// TIA Portal V20 export
FUNCTION_BLOCK "LConSMC_LevelControl"   // FB32023, SCL
// Dieser Funktionsbaustein überwacht einen Eingabewert (x), um zu erkennen ob er einen parametrierten Wert verletzt (überschreitet, unterschreitet). Der Funktionsbaustein kann in jedem zyklischen Interrupt aufgerufen werden.  Funktionsbaustein-ID: 0104 / Limit value monitor. The function block can be called in any cyclic task.  Function block ID: 0104
// stored: Access Published, IsIECCheckEnabled true, MemoryReserve 100, SetENOAutomatically true
   VAR_INPUT
      run { ExternalAccessible := 'False'; ExternalVisible := 'False'; ExternalWritable := 'False'} : Bool := FALSE;   // TRUE: Funktionsbaustein aktivieren / TRUE: Enable function block
      x { ExternalAccessible := 'False'; ExternalVisible := 'False'; ExternalWritable := 'False'} : LReal := 0.0;   // Eingangswert / Input value
      alarmHigh { ExternalAccessible := 'False'; ExternalVisible := 'False'; ExternalWritable := 'False'} : LReal := 100.0;   // Alarm, oberer Grenzwert / Alarm, upper limit value
      warningHigh { ExternalAccessible := 'False'; ExternalVisible := 'False'; ExternalWritable := 'False'} : LReal := 80.0;   // Warnung, oberer Grenzwert / Warning, upper limit value
      warningLow { ExternalAccessible := 'False'; ExternalVisible := 'False'; ExternalWritable := 'False'} : LReal := -80.0;   // Warnung, unterer Grenzwert / Warning, lower limit value
      alarmLow { ExternalAccessible := 'False'; ExternalVisible := 'False'; ExternalWritable := 'False'} : LReal := -100.0;   // Alarm, unterer Grenzwert / Alarm, lower limit value
      hyst { ExternalAccessible := 'False'; ExternalVisible := 'False'; ExternalWritable := 'False'} : LReal := 0.0;   // Hysterese (Betrag wird verwendet) / Hysteresis (Absolute value is used)
      delayTime { ExternalAccessible := 'False'; ExternalVisible := 'False'; ExternalWritable := 'False'} : Time := T#3S;   // [s] Ausgangsverzögerungszeit Für einen Wert von 0 ist die Verzögerung deaktiviert / [ s ] Output delay time delayTime = 0, signal delay is disabled
   END_VAR
   VAR_OUTPUT
      busy { ExternalAccessible := 'False'; ExternalVisible := 'False'; ExternalWritable := 'False'} : Bool := FALSE;   // TRUE: Der Funktionsbaustein ist aktiv / TRUE: Function block is activated
      alarmUpperLimit { ExternalAccessible := 'False'; ExternalVisible := 'False'; ExternalWritable := 'False'} : Bool;   // TRUE: oberer Alarmwert überschritten / TRUE: Upper alarm limit value exceeded
      alarmLowerLimit { ExternalAccessible := 'False'; ExternalVisible := 'False'; ExternalWritable := 'False'} : Bool;   // TRUE: unterer Alarmwert überschritten / TRUE: Lower alarm limit value exceeded
      warningUpperLimit { ExternalAccessible := 'False'; ExternalVisible := 'False'; ExternalWritable := 'False'} : Bool := FALSE;   // TRUE: oberer Warnwert überschritten / TRUE: Upper warning limit value exceeded
      warningLowerLimit { ExternalAccessible := 'False'; ExternalVisible := 'False'; ExternalWritable := 'False'} : Bool := FALSE;   // TRUE: unterer Warnwert überschritten / TRUE: Lower warning limit value exceeded
   END_VAR
   VAR
      statAlarmUpperLimitSafe { ExternalAccessible := 'False'; ExternalVisible := 'False'; ExternalWritable := 'False'} : Bool := FALSE;
      statWarningUpperLimitSafe { ExternalAccessible := 'False'; ExternalVisible := 'False'; ExternalWritable := 'False'} : Bool := FALSE;
      statWarningLowerLimitSafe { ExternalAccessible := 'False'; ExternalVisible := 'False'; ExternalWritable := 'False'} : Bool := FALSE;
      statAlarmLowerLimitSafe { ExternalAccessible := 'False'; ExternalVisible := 'False'; ExternalWritable := 'False'} : Bool := FALSE;
      instTONalUp { ExternalAccessible := 'False'; ExternalVisible := 'False'; ExternalWritable := 'False'} : TON_TIME;
      instTONwaUp { ExternalAccessible := 'False'; ExternalVisible := 'False'; ExternalWritable := 'False'} : TON_TIME;
      instTONwaLo { ExternalAccessible := 'False'; ExternalVisible := 'False'; ExternalWritable := 'False'} : TON_TIME;
      instTONalLo { ExternalAccessible := 'False'; ExternalVisible := 'False'; ExternalWritable := 'False'} : TON_TIME;
      statAlarmUpperLimit { ExternalAccessible := 'False'; ExternalVisible := 'False'; ExternalWritable := 'False'} : Bool := FALSE;
      statAlarmLowerLimit { ExternalAccessible := 'False'; ExternalVisible := 'False'; ExternalWritable := 'False'} : Bool := FALSE;
      statWarningUpperLimit { ExternalAccessible := 'False'; ExternalVisible := 'False'; ExternalWritable := 'False'} : Bool := FALSE;
      statWarningLowerLimit { ExternalAccessible := 'False'; ExternalVisible := 'False'; ExternalWritable := 'False'} : Bool := FALSE;
   END_VAR
BEGIN
   REGION BLOCK INFO HEADER
     //===============================================================================
     // SIEMENS AG / (c)Copyright 2023
     //-------------------------------------------------------------------------------
     // Title:            LConSMC_LevelControl
     // Comment/Function: Limit value evaluation with warning level and alarm level
     // Library/Family:   LConSMC
     // Author:           APC Erlangen
     // Tested with:      FW 2.8
     // Engineering:      TIA Portal V16
     // Restrictions:     Needs to be called in a cyclic task
     // Requirements:     -
     //-------------------------------------------------------------------------------
     // Change log table:
     // Version  | Date       | Expert in charge       | Changes applied
     //----------|------------|------------------------|------------------------------
     // 01.01.00 | 2016-11-17 | APC Erlangen           | adapted to styleguide; warning "variable might not be initialized" removed
     // 01.00.00 | 2012-07-23 | APC Erlangen           | Creation
     //===============================================================================
     //
   END_REGION BLOCK INFO HEADER

   REGION DESCRIPTION
   (/*This function block monitors an input value (x) to identify whether it violates (exceeds, falls below) parameterized limit values as long as it is active with run = TRUE.
   If the block is enabled, then this can be identified using the busy output.
   When the warningHigh value is exceeded, output warningUpperLimit is set after the delayTime.
   The same applies when the alarmHigh value is exceeded with the associated output alarmUpperLimit.
   If the input value drops below the limit value warningHigh or alarmHigh minus the hysteresis value (hyst), the particular output is reset.
   The same applies for the lower limit monitoring with the limits warningLow and alarmLow as well as the associated outputs warningLowerLimit and alarmLowerLimit.
   However, in this case, the hysteresis (hyst) is added to the limit value. 
   Warnings are not reset as a result of alarms.

   ![Level control diagram](LevelControl_Diagram.png)*/)
   END_REGION

   #busy := #run;

   // UPPER LIMIT ALARM EVALUATION
   #statAlarmUpperLimitSafe := (#run) AND
   ((#x > #alarmHigh) OR
   ((#statAlarmUpperLimit) AND (#x > #alarmHigh - ABS(#hyst))));
   #instTONalUp(IN := #statAlarmUpperLimitSafe,
                PT := #delayTime);
   #statAlarmUpperLimit := #instTONalUp.Q;

   // UPPER LIMIT WARNING EVALUATION
   #statWarningUpperLimitSafe := (#run) AND
   ((#x > #warningHigh) OR
   ((#statWarningUpperLimit) AND (#x > #warningHigh - ABS(#hyst))));
   #instTONwaUp(IN := #statWarningUpperLimitSafe,
                PT := #delayTime);
   #statWarningUpperLimit := #instTONwaUp.Q;


   // LOWER LIMIT WARNING EVALUATION
   #statWarningLowerLimitSafe := (#run) AND
   ((#x < #warningLow) OR
   ((#statWarningLowerLimit) AND (#x < #warningLow + ABS(#hyst))));

   #instTONwaLo(IN := #statWarningLowerLimitSafe,
                PT := #delayTime);
   #statWarningLowerLimit := #instTONwaLo.Q;

   // LOWER LIMIT ALARM  EVALUATION
   #statAlarmLowerLimitSafe := (#run) AND
   ((#x < #alarmLow) OR
   ((#statAlarmLowerLimit) AND (#x < #alarmLow + ABS(#hyst))));

   #instTONalLo(IN := #statAlarmLowerLimitSafe,
                PT := #delayTime);
   #statAlarmLowerLimit := #instTONalLo.Q;

   // set outputs
   #alarmUpperLimit := #statAlarmUpperLimit;
   #alarmLowerLimit := #statAlarmLowerLimit;
   #warningUpperLimit := #statWarningUpperLimit;
   #warningLowerLimit := #statWarningLowerLimit;
END_FUNCTION_BLOCK
